FUNCTION_BLOCK Produce (* Basic Function Block Type *)
  (* Standard: 61499-2 *)
  (* Version 0.0, 9/26/2018, dmidro, nxtControl GmbH, Template *)
  PACKAGE Main;
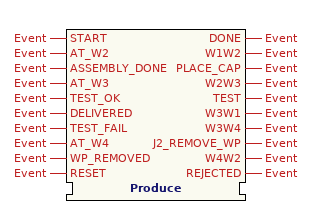
  EVENT_INPUT
    START;
    AT_W2;
    ASSEMBLY_DONE;
    AT_W3;
    TEST_OK;
    DELIVERED;
    TEST_FAIL;
    AT_W4;
    WP_REMOVED;
    RESET;
  END_EVENT
  EVENT_OUTPUT
    DONE;
    W1W2;
    PLACE_CAP;
    W2W3;
    TEST;
    W3W1;
    W3W4;
    J2_REMOVE_WP;
    W4W2;
    REJECTED;
  END_EVENT
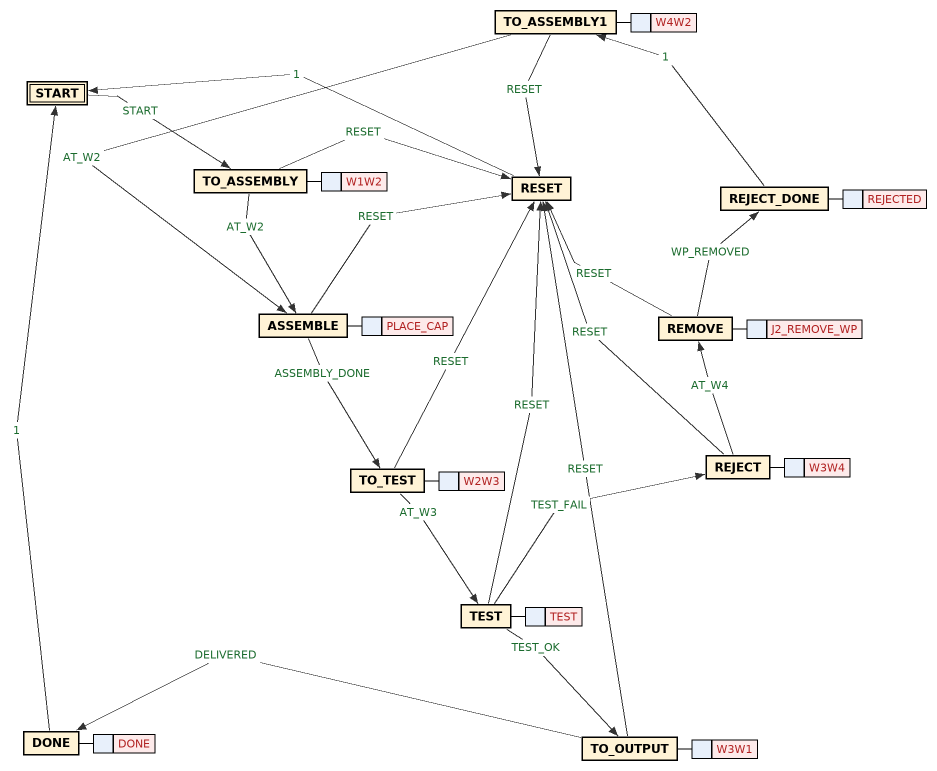
  EC_STATES
    START; (* Initial State *)
    TO_ASSEMBLY : -> W1W2;
    ASSEMBLE : -> PLACE_CAP;
    TO_TEST : -> W2W3;
    TEST : -> TEST;
    TO_OUTPUT : -> W3W1;
    DONE : -> DONE;
    REJECT : -> W3W4;
    REMOVE : -> J2_REMOVE_WP;
    REJECT_DONE : -> REJECTED;
    RESET;
    TO_ASSEMBLY1 : -> W4W2;
  END_STATES
  EC_TRANSITIONS
    START TO TO_ASSEMBLY := START;
    TO_ASSEMBLY TO ASSEMBLE := AT_W2;
    ASSEMBLE TO TO_TEST := ASSEMBLY_DONE;
    TO_TEST TO TEST := AT_W3;
    TEST TO TO_OUTPUT := TEST_OK;
    TO_OUTPUT TO DONE := DELIVERED;
    DONE TO START := 1;
    TEST TO REJECT := TEST_FAIL;
    REJECT TO REMOVE := AT_W4;
    REMOVE TO REJECT_DONE := WP_REMOVED;
    REJECT_DONE TO TO_ASSEMBLY1 := 1;
    TO_ASSEMBLY TO RESET := RESET;
    ASSEMBLE TO RESET := RESET;
    TO_TEST TO RESET := RESET;
    TEST TO RESET := RESET;
    TO_OUTPUT TO RESET := RESET;
    REJECT TO RESET := RESET;
    REMOVE TO RESET := RESET;
    RESET TO START := 1;
    TO_ASSEMBLY1 TO ASSEMBLE := AT_W2;
    TO_ASSEMBLY1 TO RESET := RESET;
  END_TRANSITIONS
  ALGORITHM INIT IN ST: (* Initialization algorithm *)
;
  END_ALGORITHM
  ALGORITHM REQ IN ST: (* Normally executed algorithm *)
;
  END_ALGORITHM
END_FUNCTION_BLOCK
